(* PLC project Unbenannt, Unbekannt Unbenannt 1 *)
(* stored: creationDateTime 2024-12-11T18:09:29, modificationDateTime 2024-12-12T16:49:51 *)

PROGRAM program0
  VAR
    sensor_0 AT %IX100.0 : BOOL;
    sensor_1 AT %IX100.1 : BOOL;
    arm_detect AT %IX100.2 : BOOL;
    motor_0 AT %QX100.0 : BOOL := True;
    motor_1 AT %QX100.1 : BOOL := True;
    motor_2 AT %QX100.2 : BOOL := True;
    motor_3 AT %QX100.3 : BOOL := True;
    arm_Z AT %QX100.4 : BOOL := False;
    arm_X AT %QX100.5 : BOOL := False;
    arm_suck AT %QX100.6 : BOOL := False;
  END_VAR
  VAR
    CL : INT := 0;
    TON0 : TON;
    TON1 : TON;
    TON2 : TON;
    TON3 : TON;
    TON4 : TON;
    TON5 : TON;
    TON6 : TON;
  END_VAR
  VAR  (* added by the conversion: wires and edge detectors of the diagram *)
    _EQ40_OUT : BOOL;
    _EQ9_ENO : BOOL;
    _EQ9_OUT : BOOL;
    _EQ18_ENO : BOOL;
    _EQ18_OUT : BOOL;
    _EQ31_ENO : BOOL;
    _EQ31_OUT : BOOL;
    _EQ49_ENO : BOOL;
    _EQ49_OUT : BOOL;
    _EQ63_ENO : BOOL;
    _EQ63_OUT : BOOL;
  END_VAR

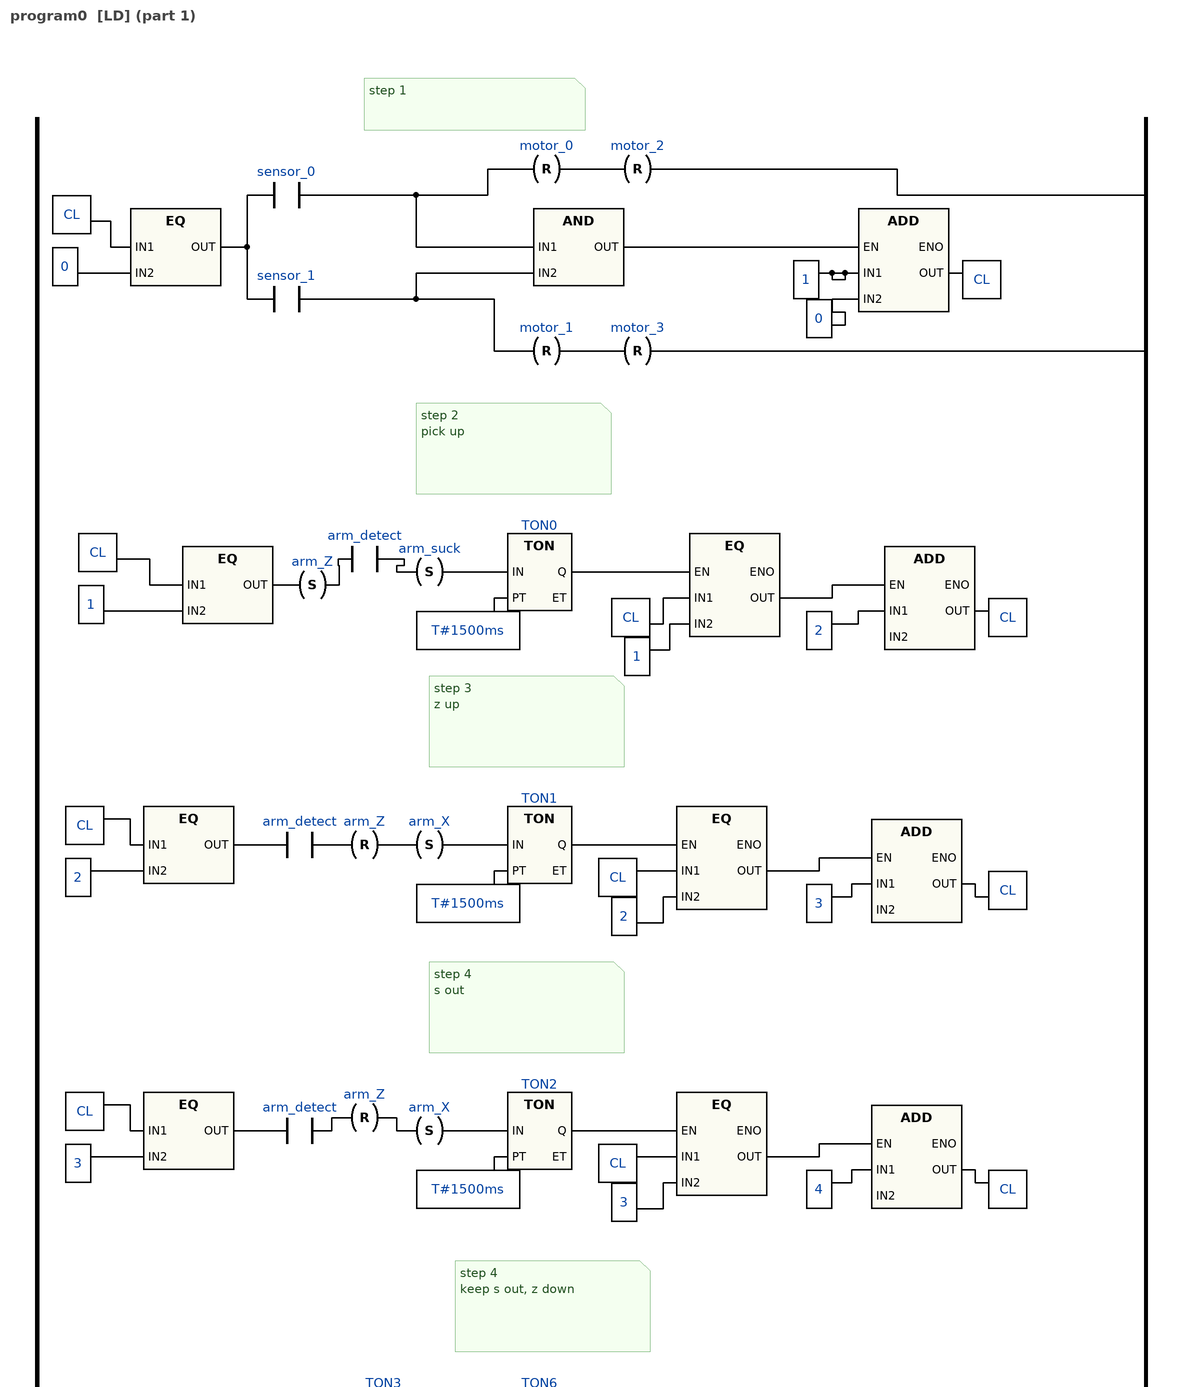
(* LD diagram, written out as Structured Text *)
(* step 1 *)
_EQ40_OUT := CL = 0;
IF _EQ40_OUT AND sensor_0 THEN motor_0 := FALSE; END_IF;
IF _EQ40_OUT AND sensor_1 THEN motor_1 := FALSE; END_IF;
IF _EQ40_OUT AND sensor_0 AND _EQ40_OUT AND sensor_1 THEN CL := 1 + 0; END_IF;
(* step 2
pick up *)
TON0(IN := CL = 1 AND arm_detect, PT := T#1500ms);
_EQ9_OUT := EQ(EN := TON0.Q, IN1 := CL, IN2 := 1, ENO => _EQ9_ENO);
IF _EQ9_OUT THEN CL := ADD(IN1 := 2); END_IF;
IF CL = 1 THEN arm_Z := TRUE; END_IF;
IF CL = 1 AND arm_detect THEN arm_suck := TRUE; END_IF;
(* step 3
z up *)
IF CL = 2 AND arm_detect THEN arm_Z := FALSE; END_IF;
TON1(IN := CL = 2 AND arm_detect, PT := T#1500ms);
_EQ18_OUT := EQ(EN := TON1.Q, IN1 := CL, IN2 := 2, ENO => _EQ18_ENO);
IF _EQ18_OUT THEN CL := ADD(IN1 := 3); END_IF;
IF CL = 2 AND arm_detect THEN arm_X := TRUE; END_IF;
(* step 4
s out *)
IF CL = 3 AND arm_detect THEN arm_Z := FALSE; END_IF;
TON2(IN := CL = 3 AND arm_detect, PT := T#1500ms);
_EQ31_OUT := EQ(EN := TON2.Q, IN1 := CL, IN2 := 3, ENO => _EQ31_ENO);
IF _EQ31_OUT THEN CL := ADD(IN1 := 4); END_IF;
IF CL = 3 AND arm_detect THEN arm_X := TRUE; END_IF;
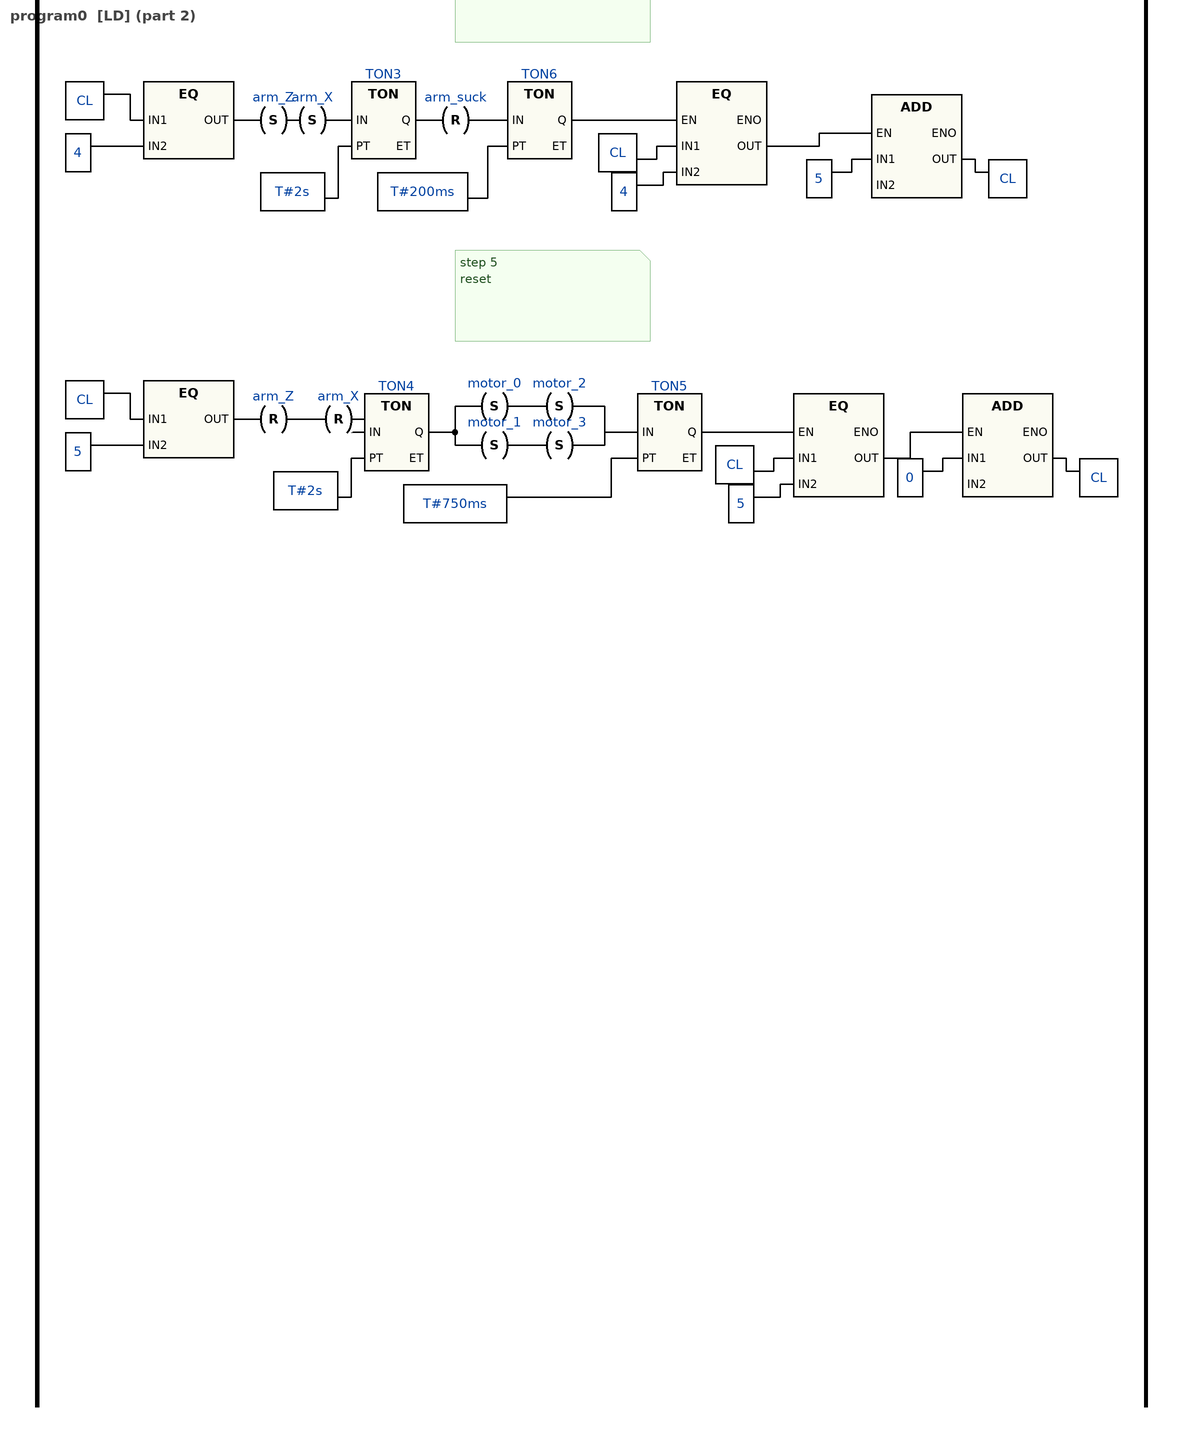
(* step 4
keep s out, z down *)
IF CL = 4 THEN arm_Z := TRUE; END_IF;
IF CL = 4 THEN arm_X := TRUE; END_IF;
TON3(IN := CL = 4, PT := T#2s);
TON6(IN := TON3.Q, PT := T#200ms);
_EQ49_OUT := EQ(EN := TON6.Q, IN1 := CL, IN2 := 4, ENO => _EQ49_ENO);
IF _EQ49_OUT THEN CL := ADD(IN1 := 5); END_IF;
IF TON3.Q THEN arm_suck := FALSE; END_IF;
(* step 5
reset *)
IF CL = 5 THEN arm_Z := FALSE; END_IF;
IF CL = 5 THEN arm_X := FALSE; END_IF;
TON4(IN := CL = 5, PT := T#2s);
TON5(IN := TON4.Q, PT := T#750ms);
_EQ63_OUT := EQ(EN := TON5.Q, IN1 := CL, IN2 := 5, ENO => _EQ63_ENO);
IF _EQ63_OUT THEN CL := ADD(IN1 := 0); END_IF;
IF _EQ40_OUT AND sensor_0 THEN motor_2 := FALSE; END_IF;
IF _EQ40_OUT AND sensor_1 THEN motor_3 := FALSE; END_IF;
IF TON4.Q THEN motor_0 := TRUE; END_IF;
IF TON4.Q THEN motor_2 := TRUE; END_IF;
IF TON4.Q THEN motor_1 := TRUE; END_IF;
IF TON4.Q THEN motor_3 := TRUE; END_IF;
END_PROGRAM

CONFIGURATION Config0
  RESOURCE Res0 ON PLC
    TASK task0(INTERVAL := T#20ms, PRIORITY := 0);
    PROGRAM instance0 WITH task0 : program0;
  END_RESOURCE
END_CONFIGURATION
